FUNCTION_BLOCK S5_AerateTime2 (* Basic Function Block Type *)
  (* Standard: 61499-2 *)
  (* Version 0.0, 7/5/2026, Schneider Electric, Template *)
  PACKAGE SE.Nereda;
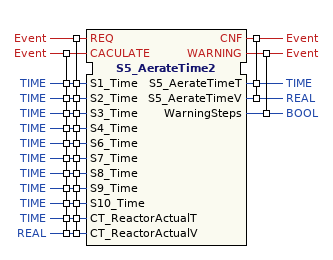
  EVENT_INPUT
    REQ WITH S1_Time, S2_Time, S3_Time, S4_Time, S6_Time, S7_Time, S8_Time, CT_ReactorActualT, CT_ReactorActualV, S9_Time, S10_Time; (* Normal Execution Request *)
    CACULATE WITH S1_Time, S2_Time, S3_Time, S4_Time, S6_Time, S7_Time, S8_Time, CT_ReactorActualT, CT_ReactorActualV, S9_Time, S10_Time;
  END_EVENT
  EVENT_OUTPUT
    CNF WITH S5_AerateTimeT, S5_AerateTimeV; (* Execution Confirmation *)
    WARNING WITH WarningSteps;
  END_EVENT
  VAR_INPUT
    S1_Time : TIME;
    S2_Time : TIME;
    S3_Time : TIME;
    S4_Time : TIME;
    S6_Time : TIME;
    S7_Time : TIME;
    S8_Time : TIME;
    S9_Time : TIME;
    S10_Time : TIME;
    CT_ReactorActualT : TIME;
    CT_ReactorActualV : REAL;
  END_VAR
  VAR_OUTPUT
    S5_AerateTimeT : TIME; (* Output event qualifier *)
    S5_AerateTimeV : REAL;
    WarningSteps : BOOL;
  END_VAR
  VAR
    InS1_Time : REAL;
    InS2_Time : REAL;
    InS3_Time : REAL;
    InS4_Time : REAL;
    InS6_Time : REAL;
    InS7_Time : REAL;
    InS8_Time : REAL;
    InS9_Time : REAL;
    InS10_Time : REAL;
    SumSteps : REAL;
  END_VAR
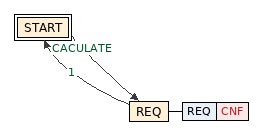
  EC_STATES
    START; (* Initial State *)
    REQ : REQ -> CNF; (* Normal execution *)
  END_STATES
  EC_TRANSITIONS
    START TO REQ := CACULATE;
    REQ TO START := 1;
  END_TRANSITIONS
  ALGORITHM REQ IN ST: (* Normally executed algorithm *)
InS1_Time := TIME_TO_REAL(S1_Time);
InS2_Time := TIME_TO_REAL(S2_Time);
InS3_Time := TIME_TO_REAL(S3_Time);
InS4_Time := TIME_TO_REAL(S4_Time);
InS6_Time := TIME_TO_REAL(S6_Time);
InS7_Time := TIME_TO_REAL(S7_Time);
InS8_Time := TIME_TO_REAL(S8_Time);
InS9_Time := TIME_TO_REAL(S9_Time);
InS10_Time := TIME_TO_REAL(S10_Time);
SumSteps := InS1_Time + InS2_Time + InS3_Time + InS4_Time + InS6_Time + InS7_Time + InS8_Time + InS9_Time + InS10_Time;

S5_AerateTimeV := CT_ReactorActualV - SumSteps;

IF S5_AerateTimeV < 0 THEN
	WarningSteps := TRUE;
	S5_AerateTimeV := 0;
	S5_AerateTimeT := T#0s;
ELSE
	WarningSteps := FALSE;
	S5_AerateTimeT := REAL_TO_TIME(S5_AerateTimeV);
END_IF;
  END_ALGORITHM
END_FUNCTION_BLOCK
